FUNCTION_BLOCK FB_SigCond_MovingAverage
VAR_INPUT
	fIn:					FLOAT;
	nSamplesToFilter:		UINT; // Maximum of 500
	tCtrlCycleTime:			TIME;
	tTaskCycleTime:			TIME;

	fManSyncValue:	FLOAT;
	bSync:			BOOL;
	eMode:			E_CTRL_MODE;
	bHold:			BOOL;
END_VAR

VAR
	
	fbCtr_MovAvg:	FB_CTRL_MOVING_AVERAGE;
	stParams:		ST_CTRL_MOVING_AVERAGE_PARAMS;
	aInternalData:	ARRAY[1..500] OF FLOAT;
END_VAR


VAR_OUTPUT
	fOut:			FLOAT;
	eState:			E_CTRL_STATE;
	eErrorID:		E_CTRL_ERRORCODES;
	bError:			BOOL;	
END_VAR



// Read inputs and put into params structure
stParams.nSamplesToFilter 	:= nSamplesToFilter;
stParams.tCtrlCycleTime 	:= tCtrlCycleTime;
stParams.tTaskCycleTime		:= tTaskCycleTime;
stParams.pWorkArray_ADR		:= ADR(aInternalData);
stParams.nWorkArray_SIZEOF	:= SIZEOF(aInternalData);

eMode := E_CTRL_MODE.eCTRL_MODE_ACTIVE;

// Execute filter
fbCtr_MovAvg(fIn := fIn, fManSyncValue := fManSyncValue, bSync := bSync, eMode := eMode, bHold := bHold, stParams := stParams);


// Update outputs
fOut 		:= fbCtr_MovAvg.fOut;
eState 		:= fbCtr_MovAvg.eState;
eErrorID 	:= fbCtr_MovAvg.eErrorId;
bError 		:= fbCtr_MovAvg.bError;

END_FUNCTION_BLOCK

(* stored: Version 1.1.0.1, ProductVersion 3.1.4024.12
   POU FB_SigCond_MovingAverage: Id {3bb2ebc7-4f34-432f-ba5d-d27d2db361ff}, SpecialFunc None *)
